FUNCTION_BLOCK FB_Shelly_3EM
VAR_INPUT
	bStart				: BOOL;
	tDelayRequest		: TIME;		//Timer for delay before start with the next read or write Request
	sHostname			: STRING(255);		//Hostname or IP Adress from the Server
END_VAR

VAR_IN_OUT
END_VAR

VAR_OUTPUT
	bValidResult		: BOOL;							//Valid Result received from Server
    bBusy				: BOOL;							//Function is Busy
    bError				: BOOL;							//Error sucess
	bDone				: BOOL;							//True after the decoding from the received Json File
	bConnected			: BOOL;							//Connection to the Server
	lrtotalpower		: LREAL;						//Received Value
	lrpowerL1			: LREAL;
	lrcurrentL1			: LREAL;
	lrvoltageL1			: LREAL;
	lrenergyL1			: LREAL;
	lrpowerL2			: LREAL;
	lrcurrentL2			: LREAL;
	lrvoltageL2			: LREAL;
	lrenergyL2			: LREAL;
	lrpowerL3			: LREAL;
	lrcurrentL3			: LREAL;
	lrvoltageL3			: LREAL;
	lrenergyL3			: LREAL;
	hrErrorCode       	: HRESULT;						//Error Result from Http Client
END_VAR

VAR
	fbClient			: FB_IotHttpClient;
	fbHttpGet			: FB_Shelly_3EM_Helper;
	timStartRequest		: TON;							//Timer to Start the Request
	FPStartRequest		: R_TRIG;						//Internal positive Edge
	FPDone				: R_TRIG;						//Internal positive Edge
	FNStart				: F_TRIG;						//Internal negative Edge
	y: INT;
END_VAR

(*------------------------------------------------------------------------------------Configure HTTP Client------------------------------------------------------------------------------------------------------*)

fbClient.sHostName := sHostname;
fbClient.tConnectionTimeout := T#30S;

IF NOT fbClient.bConfigured THEN 
	fbClient.nHostPort:= 80;
	fbClient.bKeepAlive := TRUE;
	fbClient.tConnectionTimeout := T#30S;
END_IF


//Timer to start the Request
FPStartRequest(CLK:= bStart, Q=> );
timStartRequest(IN:= fbClient.bConfigured AND bStart AND NOT timStartRequest.Q, PT:= tDelayRequest, Q=> , ET=> );

IF ((timStartRequest.Q AND NOT bBusy) OR (FPStartRequest.Q AND NOT bBusy AND fbClient.bConfigured)) THEN 
	y:=y+1;
	fbHttpGet.bSend := TRUE; 
END_IF

				
//Http Get Function
fbHttpGet(
	lrtotalpower => lrtotalpower, 
	lrpowerL1 => lrpowerL1,
	lrcurrentL1 => lrcurrentL1,
	lrvoltageL1 => lrvoltageL1,
	lrenergyL1 => lrenergyL1,
	lrpowerL2 => lrpowerL2,
	lrcurrentL2 => lrcurrentL2,
	lrvoltageL2 => lrvoltageL2,
	lrenergyL2 => lrenergyL2,
	lrpowerL3 => lrpowerL3,
	lrcurrentL3 => lrcurrentL3,
	lrvoltageL3 => lrvoltageL3,
	lrenergyL3 => lrenergyL3,
	bSend:= , 
	fbClient:= fbClient, 
	bBusy=> bBusy, 
	bError=> ,
	sContentStatus=> ,
	sContentM0=> ,
	sContentM1=> ,
	sContentM2=> );


fbHttpGet.bSend := FALSE;

FPDone(CLK:= bDone, Q=> );

(*
//Http Client
FNStart(CLK:= bStart, Q=> );
	IF FNStart.Q THEN fbClient.Disconnect(); END_IF
*)

fbClient.Execute();

//Error
IF fbHttpGet.bError OR fbClient.bError THEN 
	bError := TRUE; 
ELSE 
	bError := FALSE; 
END_IF	

hrErrorCode := fbClient.hrErrorCode;

END_FUNCTION_BLOCK

(* stored: Version 1.1.0.1, ProductVersion 3.1.4024.11
   POU FB_Shelly_3EM: Id {85fd4c6b-d2c3-4a9a-847e-fab824f86deb}, SpecialFunc None *)
